PROGRAM MAIN
VAR
  LocalPermit : BOOL;
END_VAR


Plant.MixerRenamed(Start := LocalPermit);
Plant.ValveCommand := LocalPermit;

END_PROGRAM
